(* Logix 5000 project; controller cal1615 1756-L62 rev 20.19; software revision 20.05; part 81 of 81 *)
(* tags used below, declared in another part *)
   A00 : ALIAS FOR hmi_dint[0].0;
   A12 : ALIAS FOR hmi_dint[0].12;
   A30 : ALIAS FOR hmi_dint[0].30;
   acc_pos_last : REAL;
   acc_rate_dt : REAL;   // Accumulator Payout Rate Sample Interval Guarded Scan Time [s]
   acc_rate_meas : REAL;
   acc_rate_raw : REAL;
   acc_rate_target : REAL;
   acc_taper : REAL;
   add_sys_ramp : sys_Ramp;   // Addon Ramp
   ai_lpt01_pct : REAL;   // AI: Linear Position Transducer [%]
   ao_prs01 : REAL;   // AO: Pressure 1
   ao_prs02 : REAL;   // AO: Pressure 2
   control_to_empty : ALIAS FOR hmi_dint[9].13;
   di_ss_close_nip : ALIAS FOR p00_io_winder:5:I.14;
   di_ss_nip_auto : ALIAS FOR p00_io_winder:5:I.13;
   do_carriage_lift_sol : ALIAS FOR p00_io_winder:4:O.7;
   do_close_nip_sol : ALIAS FOR p00_io_winder:4:O.8;
   do_nip_illuminated_ss : ALIAS FOR p00_io_winder:4:O.6;
   enable_control : BOOL;   // Accumulator - Enable Control
   Me : ALIAS FOR p00_wac;
   nip_auto_open_request : BOOL;   // Nip Auto Open Request
   nip_close_request : ALIAS FOR hmi_dint[9].7;
   nip_mode_auto : BOOL;   // Nip Mode Auto
   nip_open_dwell : TIMER;   // Nip Roll Open Dwell Payout must be established before the nip lets go
   nip_open_request : BOOL;   // Nip Open Request
   nip_open_selected : BOOL;   // Nip Selector in OPEN Neither Auto nor Close
   oneshot : DINT;
   param_acc_capacity_ft : REAL;   // Parameter Accumulator Web Capacity at Full Stroke 26 s at 23 fpm measured [ft]
   param_acc_empty_hyst : REAL;
   param_acc_empty_pct : REAL;
   param_acc_min_limit : REAL;   // Parameter Accumulator Low Min Limimt
   param_acc_taper_pct : REAL;
   param_accel_rate : REAL;   // Parameter Acceleration Rate
   param_counter_prs : REAL;   // Parameter Counter Pressure
   param_decel_rate : REAL;   // Parameter Decleration Rate
   param_payout_overspeed : REAL;
   param_prs_fill : REAL;
   param_prs_payout : REAL;
   param_rate_filter : REAL;   // Parameter Accumulator Payout Rate Filter Coefficient 0.05 = about 0.4 s at a 20 ms scan
   pb_acc_on : ALIAS FOR hmi_dint[9].2;
   request_fill : ALIAS FOR hmi_dint[9].1;
   selected_pressure : REAL;   // Accumulator Selected Tension Pressure
   timer_nip_open_delay : TIMER;   // Nip Open Dwell Timer
   W00 : ALIAS FOR hmi_dint[2].0;
   FAULT : BOOL;   // Fault AFI
   HMI : BOOL;   // AFI HMI
   nip_mode_close : BOOL;   // Nip Mode Close
   p00_FlashBit_1Sec : BOOL;   // System Flash Bit 1 Second
   p00_pb_lamp_test : BOOL;
   p00_wac : Accumulator;   // Winder Accumulator
   p00_wac_enabled : BOOL;   // Winder Accumulator Enabled Carriage lift on and pressure commanded Controls which loop holds web tension
   p00_wac_position_pct : REAL;   // Winder Accumulator Carriage Position Filtered [% of Stroke]
   p00_wac_rate_error : REAL;
   p00_wac_rate_meas : REAL;
   p01r02_plc_scan_time_in_sec : REAL;   // System PLC Scan Time in Seconds
   p01r09 : routine;   // System Modes
   p01r12_master_ramped_speed : REAL;   // System Line Accel Decel Control Master Ramped Speed
   p01r12_zero_line_speed : BOOL;   // System Line Accel Decel Control Line Speed at Zero
   p29_ai_wdr_lc : REAL;   // Winder Analog Input Winder Load Cell
   p29r15_request_run : BOOL;   // Winder Winder A VFD Request Run
   p29r16_request_run : BOOL;   // Winder Winder B VFD Request Run
(* P31_WAC, continued *)

ROUTINE R11_Modes   (* ladder *)
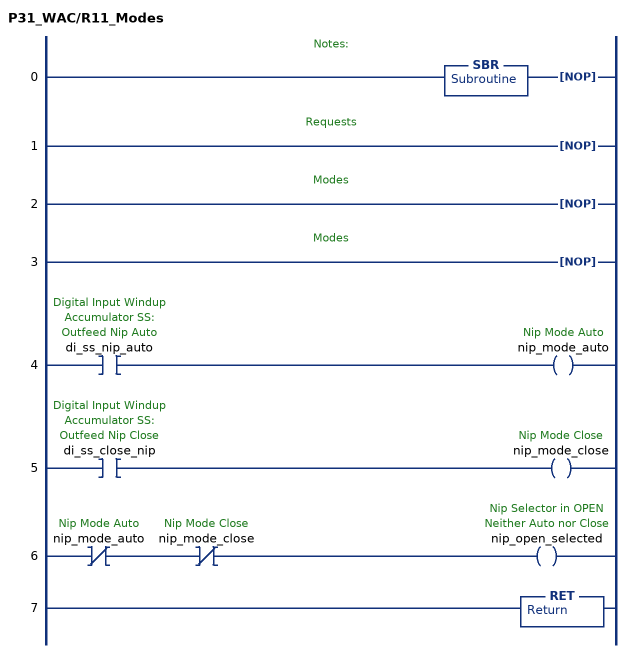
   // Notes:
   0: SBR()NOP();
   // Requests
   1: NOP();
   // Modes
   2: NOP();
   // Modes
   3: NOP();
   4: XIC(di_ss_nip_auto)OTE(nip_mode_auto);
   5: XIC(di_ss_close_nip)OTE(nip_mode_close);
   6: XIO(nip_mode_auto)XIO(nip_mode_close)OTE(nip_open_selected);
   7: RET();
END_ROUTINE

ROUTINE R21_Fill_Request   (* ladder *)
// WAC
// Fill Request and Tension Enable
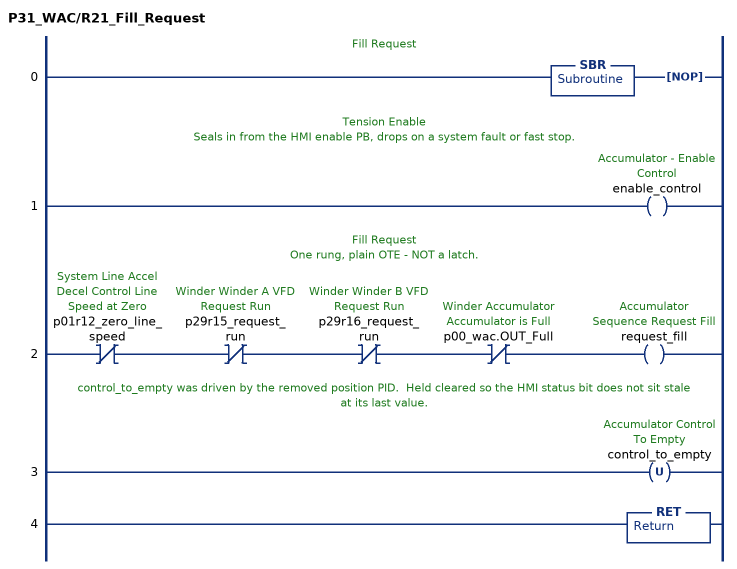
   // Fill Request
   0: SBR()NOP();
   // Tension Enable
   // Seals in from the HMI enable PB, drops on a system fault or fast stop.
   1: OTE(enable_control);
   // Fill Request
   // One rung, plain OTE - NOT a latch.
   2: XIO(p01r12_zero_line_speed)XIO(p29r15_request_run)XIO(p29r16_request_run)XIO(p00_wac.OUT_Full)OTE(request_fill);
   // control_to_empty was driven by the removed position PID.  Held cleared so the HMI status bit does not sit stale at its last value.
   3: OTU(control_to_empty);
   4: RET();
END_ROUTINE

ROUTINE R22_Fill_Pressure   (* ladder *)
// Windup Accumulator
// Fill Pressure
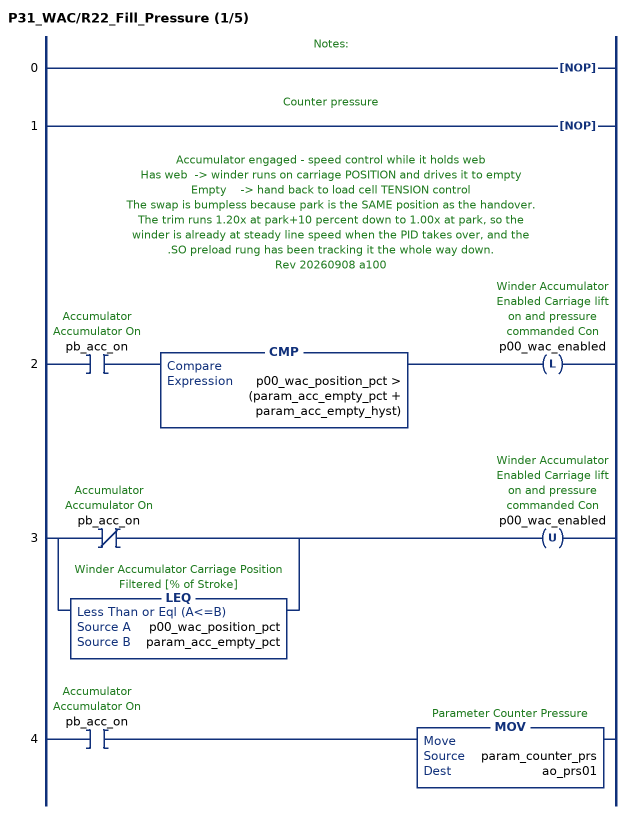
   // Notes:
   0: NOP();
   // Counter pressure
   1: NOP();
   // Accumulator engaged - speed control while it holds web
   // Has web  -> winder runs on carriage POSITION and drives it to empty
   // Empty    -> hand back to load cell TENSION control
   // The swap is bumpless because park is the SAME position as the handover.
   // The trim runs 1.20x at park+10 percent down to 1.00x at park, so the
   // winder is already at steady line speed when the PID takes over, and the
   // .SO preload rung has been tracking it the whole way down.
   // Rev 20260908 a100
   2: XIC(pb_acc_on)CMP(p00_wac_position_pct > (param_acc_empty_pct + param_acc_empty_hyst))OTL(p00_wac_enabled);
   3: [XIO(pb_acc_on) ,LEQ(p00_wac_position_pct,param_acc_empty_pct) ]OTU(p00_wac_enabled);
   4: XIC(pb_acc_on)MOV(param_counter_prs,ao_prs01);
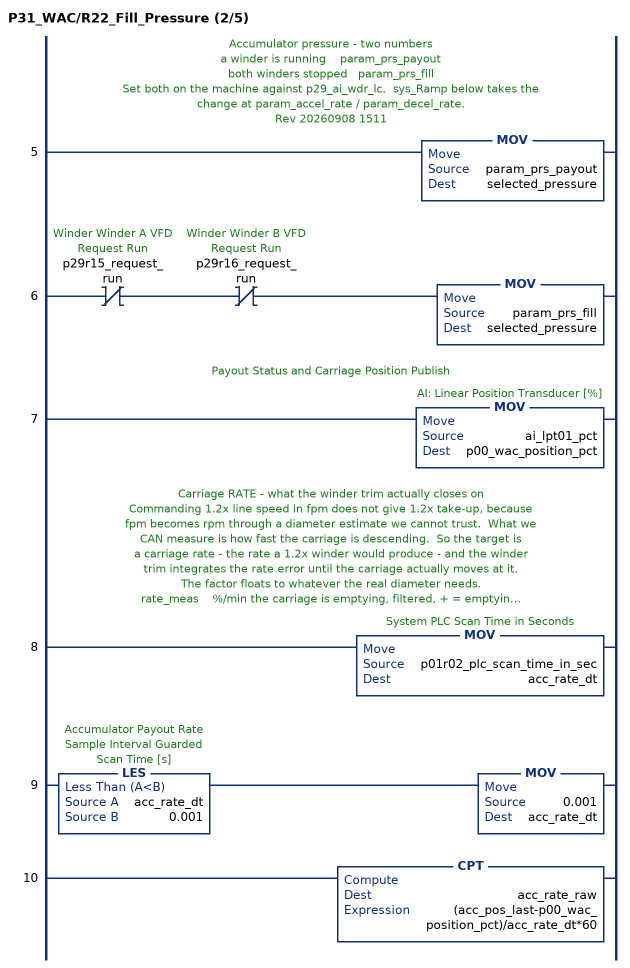
   // Accumulator pressure - two numbers
   //   a winder is running    param_prs_payout
   //   both winders stopped   param_prs_fill
   // Set both on the machine against p29_ai_wdr_lc.  sys_Ramp below takes the
   // change at param_accel_rate / param_decel_rate.
   // Rev 20260908 1511
   5: MOV(param_prs_payout,selected_pressure);
   6: XIO(p29r15_request_run)XIO(p29r16_request_run)MOV(param_prs_fill,selected_pressure);
   // Payout Status and Carriage Position Publish
   7: MOV(ai_lpt01_pct,p00_wac_position_pct);
   // Carriage RATE - what the winder trim actually closes on
   // Commanding 1.2x line speed in fpm does not give 1.2x take-up, because
   // fpm becomes rpm through a diameter estimate we cannot trust.  What we
   // CAN measure is how fast the carriage is descending.  So the target is
   // a carriage rate - the rate a 1.2x winder would produce - and the winder
   // trim integrates the rate error until the carriage actually moves at it.
   // The factor floats to whatever the real diameter needs.
   //   rate_meas    %/min the carriage is emptying, filtered, + = emptying
   //   rate_target  overspeed x line_fpm / capacity_ft x 100
   //                tapered to 0 across the last param_acc_taper_pct above
   //                the bottom, so the carriage decelerates into the stop
   //   rate_error   target - measured, integrated in P29 R10/R11
   // Rev 20260908 1514
   8: MOV(p01r02_plc_scan_time_in_sec,acc_rate_dt);
   9: LES(acc_rate_dt,0.001)MOV(0.001,acc_rate_dt);
   10: CPT(acc_rate_raw,(acc_pos_last-p00_wac_position_pct)/acc_rate_dt*60);
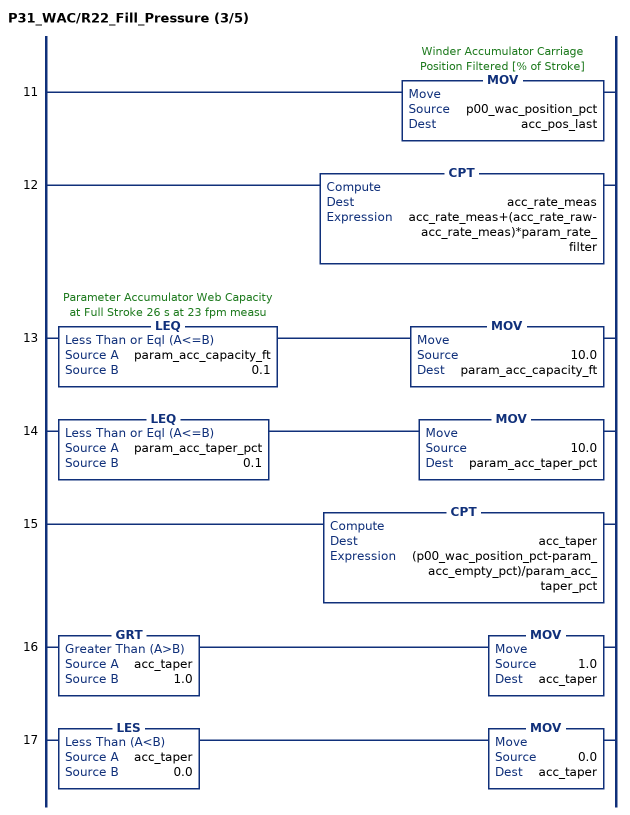
   11: MOV(p00_wac_position_pct,acc_pos_last);
   12: CPT(acc_rate_meas,acc_rate_meas+(acc_rate_raw-acc_rate_meas)*param_rate_filter);
   13: LEQ(param_acc_capacity_ft,0.1)MOV(10.0,param_acc_capacity_ft);
   14: LEQ(param_acc_taper_pct,0.1)MOV(10.0,param_acc_taper_pct);
   15: CPT(acc_taper,(p00_wac_position_pct-param_acc_empty_pct)/param_acc_taper_pct);
   16: GRT(acc_taper,1.0)MOV(1.0,acc_taper);
   17: LES(acc_taper,0.0)MOV(0.0,acc_taper);
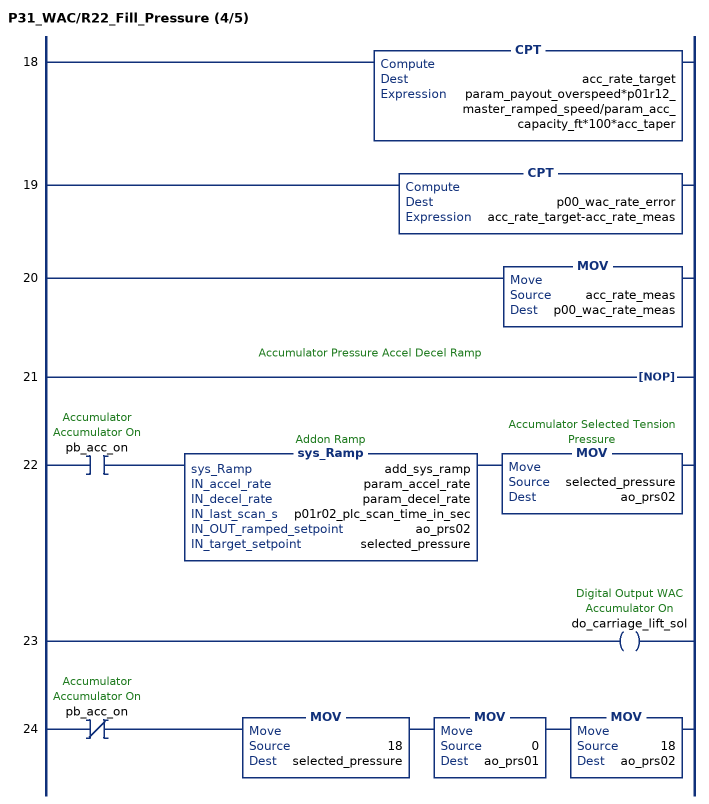
   18: CPT(acc_rate_target,param_payout_overspeed*p01r12_master_ramped_speed/param_acc_capacity_ft*100*acc_taper);
   19: CPT(p00_wac_rate_error,acc_rate_target-acc_rate_meas);
   20: MOV(acc_rate_meas,p00_wac_rate_meas);
   // Accumulator Pressure Accel Decel Ramp
   21: NOP();
   22: XIC(pb_acc_on)sys_Ramp(add_sys_ramp,param_accel_rate,param_decel_rate,p01r02_plc_scan_time_in_sec,ao_prs02,selected_pressure)MOV(selected_pressure,ao_prs02);
   23: OTE(do_carriage_lift_sol);
   24: XIO(pb_acc_on)MOV(18,selected_pressure)MOV(0,ao_prs01)MOV(18,ao_prs02);
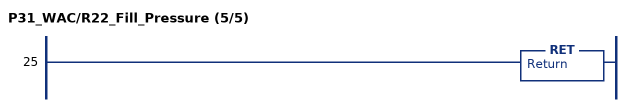
   25: RET();
END_ROUTINE

ROUTINE R31_Nip_Roll   (* ladder *)
// WAC
// Nip Roll
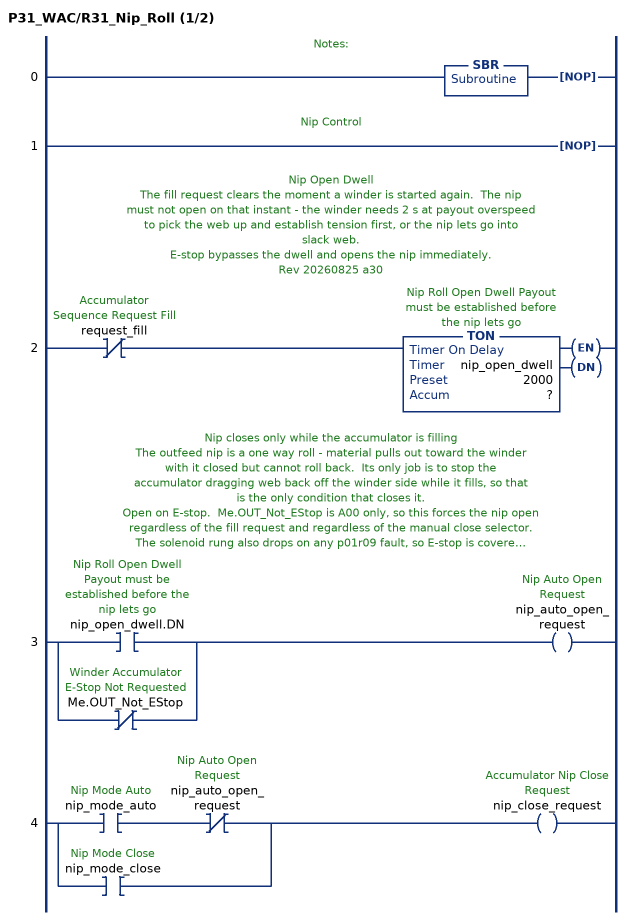
   // Notes:
   0: SBR()NOP();
   // Nip Control
   1: NOP();
   // Nip Open Dwell
   // The fill request clears the moment a winder is started again.  The nip
   // must not open on that instant - the winder needs 2 s at payout overspeed
   // to pick the web up and establish tension first, or the nip lets go into
   // slack web.
   // E-stop bypasses the dwell and opens the nip immediately.
   // Rev 20260825 a30
   2: XIO(request_fill)TON(nip_open_dwell,?,?);
   // Nip closes only while the accumulator is filling
   // The outfeed nip is a one way roll - material pulls out toward the winder
   // with it closed but cannot roll back.  Its only job is to stop the
   // accumulator dragging web back off the winder side while it fills, so that
   // is the only condition that closes it.
   // Open on E-stop.  Me.OUT_Not_EStop is A00 only, so this forces the nip open
   // regardless of the fill request and regardless of the manual close selector.
   // The solenoid rung also drops on any p01r09 fault, so E-stop is covered
   // twice - deliberately.
   // Previously opened on accumulator level above param_acc_min_limit.  That
   // left it open during the fill, which is the one time it needs to be shut.
   // No open delay - the level-based version needed one, this does not.
   // timer_nip_open_delay is left declared and unused.
   // Rev 20260825 a12
   3: [XIC(nip_open_dwell.DN) ,XIO(Me.OUT_Not_EStop) ]OTE(nip_auto_open_request);
   4: [XIC(nip_mode_auto) XIO(nip_auto_open_request) ,XIC(nip_mode_close) ]OTE(nip_close_request);
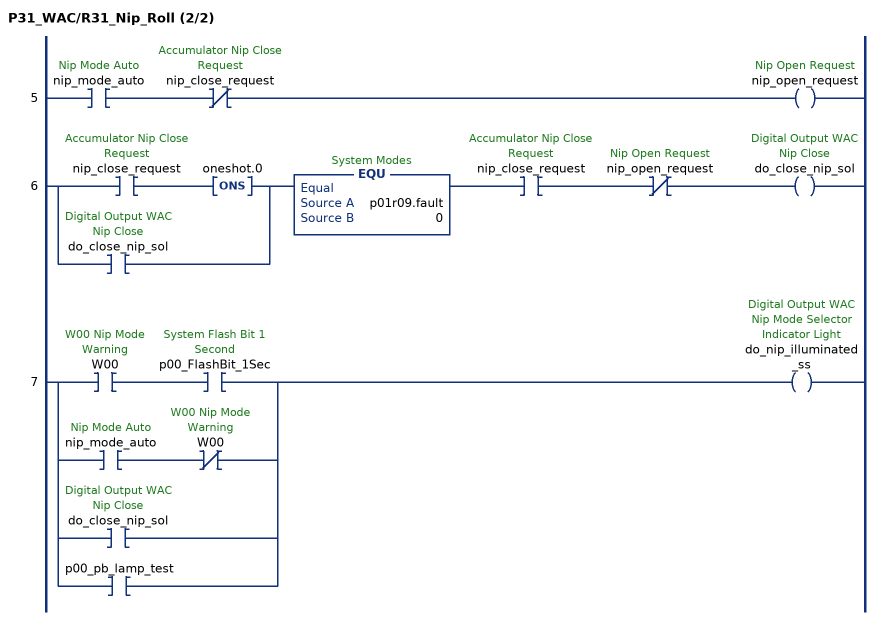
   5: XIC(nip_mode_auto)XIO(nip_close_request)OTE(nip_open_request);
   6: [XIC(nip_close_request) ONS(oneshot.0) ,XIC(do_close_nip_sol) ]EQU(p01r09.fault,0)XIC(nip_close_request)XIO(nip_open_request)OTE(do_close_nip_sol);
   7: [XIC(W00) XIC(p00_FlashBit_1Sec) ,XIC(nip_mode_auto) XIO(W00) ,XIC(do_close_nip_sol) ,XIC(p00_pb_lamp_test) ]OTE(do_nip_illuminated_ss);
END_ROUTINE
END_PROGRAM

PROGRAM ZZZ
END_PROGRAM
